// TIA Portal V18 export
DATA_BLOCK "execute_semiauto_DB"   // DB36
VERSION : 0.1
// stored: AutoNumber true, DBAccessibleFromOPCUA true, InstanceOfName execute_semiauto, InstanceOfType FB
"execute_semiauto"
   // VAR_INPUT
   //    ALLOWED : Bool;
   //    xButton : Bool;
   //    arrived : Bool;
   // END_VAR
   // VAR_OUTPUT
   //    y_exec : Bool;
   // END_VAR
   // VAR
   //    mem : Bool;
   //    R_TRIG_Instance { S7_SetPoint := 'True'} : R_TRIG;
   //    loc : Bool;
   // END_VAR
BEGIN
END_DATA_BLOCK
